// TIA Portal V20 export
TYPE "typeFeedbackFault"
// stored: Access Published, IsFailsafeCompliant true, Namespace Safety
   STRUCT
      MCFeedbackFault1 : Bool;   // Manifold1ControlPowerFeedBack
      MCFeedbackFault2 : Bool;   // Manifold2ControlPowerFeedBack
      MCFeedbackFault3 : Bool;   // FFU1ControlPowerFeedBack
      MCFeedbackFault4 : Bool;   // FFU2ControlPowerFeedBack
   END_STRUCT;
END_TYPE
